// TIA Portal V19 export
TYPE "UDT_STATUS_AIN"
   STRUCT
      fault : Bool;
      warning : Bool;
      justHadFault : Bool;
      justLostFault : Bool;
      justHadWarning : Bool;
      justLostWarning : Bool;
      value : Real;
      enabled { ExternalAccessible := 'False'; ExternalVisible := 'False'; ExternalWritable := 'False'} : Bool;
      unit : WString;
      sim : Struct
         en : Bool;
         value : Bool;
      END_STRUCT;
      old : Struct
         fault : Bool;
         warning : Bool;
      END_STRUCT;
   END_STRUCT;
END_TYPE
